{attribute 'hide_all_locals'}
{attribute 'conditionalshow'}
FUNCTION_BLOCK FB_CV_WORD_TO_LREAL_FLOAT
VAR_INPUT
	{attribute 'hide'}
	wInputValue_1				: WORD;								//Input value that is converted into the output value
	{attribute 'hide'}
	wInputValue_2				: WORD;								//Input value that is converted into the output value
	{attribute 'hide'}
	wInputValue_3				: WORD;								//Input value that is converted into the output value
	{attribute 'hide'}
	wInputValue_4				: WORD;								//Input value that is converted into the output value
	{attribute 'hide'}
	eByteOrderForConvert		: eByteOrder;						//Byte Format
END_VAR
VAR_OUTPUT
	{attribute 'hide'}
	lrOutputValue				: LREAL;							//Converted output value							
END_VAR
VAR
	unConvertLRealToULINT		: ST_UN_FLOAT_CONVERT_ULINT_LREAL;	//Union to convert the value
END_VAR

//Creator : Kai Ebensperger
//Company : Lynus AG
//Date : 28.04.2021
//Version : 1.0.0.0

//With this functionblock its possible to convert a certain Datatyp in a other Datatype
//The byte order can be selected between BigEndian and LittleEndian
//WORD TO LREAL
//Created for the Edge Device Lib over Modbus TCP
//Modbus TCP is WORD oriented

IF eByteOrderForConvert = eByteOrder.eBigEndian THEN
	unConvertLRealToULINT.uliRawValue := SHL(WORD_TO_ULINT(wInputValue_1),48) + SHL(WORD_TO_ULINT(wInputValue_2),32) + SHL(WORD_TO_ULINT(wInputValue_3),16) + WORD_TO_DWORD(wInputValue_4);
ELSE
	unConvertLRealToULINT.uliRawValue := SHL(WORD_TO_ULINT(wInputValue_4),48) + SHL(WORD_TO_ULINT(wInputValue_3),32) + SHL(WORD_TO_ULINT(wInputValue_2),16) + WORD_TO_DWORD(wInputValue_1);
END_IF

IF IsFinite(F_LREAL(unConvertLRealToULINT.lrValueFloat)) THEN
	lrOutputValue := unConvertLRealToULINT.lrValueFloat;
END_IF

END_FUNCTION_BLOCK

(* stored: Version 1.1.0.1, ProductVersion 3.1.4024.9
   POU FB_CV_WORD_TO_LREAL_FLOAT: Id {4cf9d147-3913-44c3-919a-965f59294bd2}, SpecialFunc None *)
